PROGRAM MAIN
VAR
	Power: MC_Power;
	MoveVelocity: MC_MoveVelocity;
	Halt: MC_Halt;
	ReadStatus: MC_ReadStatus;
	Timer: TON;
END_VAR

StartStopMotor();

ACTION StartStopMotor:
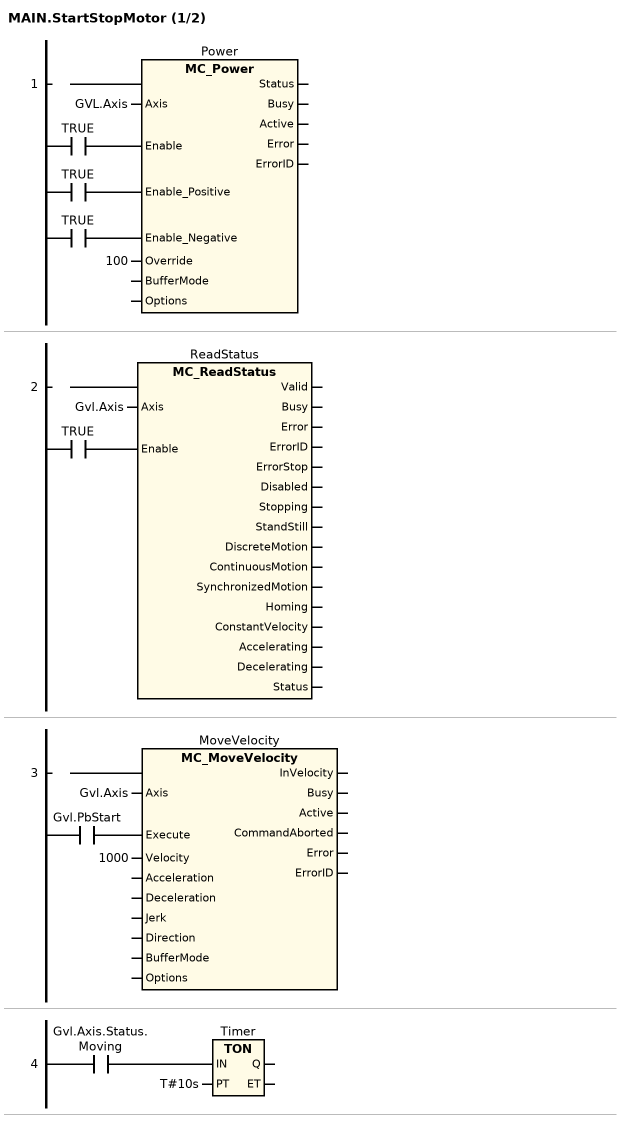
// NETWORK 1
Power(Axis := GVL.Axis, Enable := TRUE, Enable_Positive := TRUE, Enable_Negative := TRUE, Override := 100); // MC_Power

// NETWORK 2
ReadStatus(Axis := Gvl.Axis, Enable := TRUE); // MC_ReadStatus

// NETWORK 3
MoveVelocity(Axis := Gvl.Axis, Execute := Gvl.PbStart, Velocity := 1000); // MC_MoveVelocity

// NETWORK 4
Timer(IN := Gvl.Axis.Status.Moving, PT := T#10s); // TON

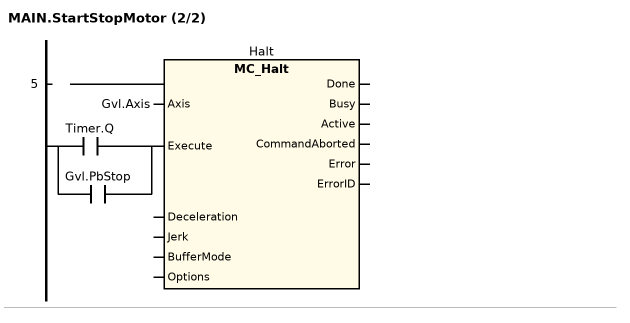
// NETWORK 5
Halt(Axis := Gvl.Axis, Execute := Timer.Q OR Gvl.PbStop); // MC_Halt
END_ACTION

END_PROGRAM

(* stored: Version 1.1.0.1, ProductVersion 3.1.4024.12
   POU MAIN: Id {43a52959-78dc-4331-a7e0-b875d8a8cbed}, SpecialFunc None
   Action StartStopMotor: Id {5069fd0f-3d49-400f-8dcc-8d657ccd3cf3} *)
